# B&R Automation Studio project PrzewijarkaBRPraktyki (part 2)

#### RecipeMenage.st
```iecst
ACTION actRecipeManage:

		//Call TableConfiguration Variable
		RecipeControl.TableControl.Config;

		// create default recipes in case they don't exist yet on the target
		// recipes are created by using the the MpRecipeXml instance interface

		CASE RecipeCreateStep OF
			IDLE:

				IF MpRecepieXml_0.Active = TRUE AND MpRecipeUI_0.Active = TRUE THEN

				RecipeCreateStep 			:= CREATE_1;

				END_IF

			CREATE_1:	// create the first recipe with default values, file name and a known picture index (Bitmap Group in the HMI)
				MpRecepieXml_0.ErrorReset 			:= FALSE;

				gHMI.Recipe.CurrentRecipe.TensionLeft := 20;
				gHMI.Recipe.CurrentRecipe.TensionRight := 20;
				gHMI.Recipe.CurrentRecipe.Speed := 4;
				gHMI.Recipe.CurrentRecipe.Dencer1PID.P := 10;
				gHMI.Recipe.CurrentRecipe.Dencer1PID.I := 1;
				gHMI.Recipe.CurrentRecipe.Dencer2PID.P := 10;
				gHMI.Recipe.CurrentRecipe.Dencer2PID.I := 1;
				gHMI.Recipe.CurrentRecipe.RollLeft.MaxSize := 80;
				gHMI.Recipe.CurrentRecipe.RollLeft.MinSize := 30;
				gHMI.Recipe.CurrentRecipe.RollRight.MaxSize := 80;
				gHMI.Recipe.CurrentRecipe.RollRight.MinSize := 30;
				gHMI.Recipe.CurrentRecipe.DataRegistration := FALSE;

				MpRecepieXml_0.FileName 				:= ADR('mappRecipe1Test.xml');
				MpRecepieXml_0.Save					:= TRUE;
				RecipeCreateStep 					:= DONE_1;

			DONE_1:	// when CommandDone GoTo next step
				IF(MpRecepieXml_0.CommandDone) THEN
					RecipeCreateStep 			:= CREATE_2;
					MpRecepieXml_0.Save			:= FALSE;
				END_IF;

			CREATE_2:	// create the next recipe with default values, file name and a known picture index (Bitmap Group in the HMI)
				gHMI.Recipe.CurrentRecipe.TensionLeft := 40;
				gHMI.Recipe.CurrentRecipe.TensionRight := 40;
				gHMI.Recipe.CurrentRecipe.Speed := 8;
				gHMI.Recipe.CurrentRecipe.Dencer1PID.P := 10;
				gHMI.Recipe.CurrentRecipe.Dencer1PID.I := 1;
				gHMI.Recipe.CurrentRecipe.Dencer2PID.P := 10;
				gHMI.Recipe.CurrentRecipe.Dencer2PID.I := 1;
				gHMI.Recipe.CurrentRecipe.RollLeft.MaxSize := 80;
				gHMI.Recipe.CurrentRecipe.RollLeft.MinSize := 30;
				gHMI.Recipe.CurrentRecipe.RollRight.MaxSize := 80;
				gHMI.Recipe.CurrentRecipe.RollRight.MinSize := 30;
				gHMI.Recipe.CurrentRecipe.DataRegistration := FALSE;

				MpRecepieXml_0.FileName 			:= ADR('mappRecipe2Test.xml');
				MpRecepieXml_0.Save					:= TRUE;
				RecipeCreateStep 					:= DONE_2;

			DONE_2:	// when CommandDone GoTo next step
				IF (MpRecepieXml_0.CommandDone) THEN
					RecipeCreateStep 			:= CREATE_3;
					MpRecepieXml_0.Save			:= FALSE;
				END_IF;

			CREATE_3:	// create the next recipe with default values, file name and a known picture index (Bitmap Group in the HMI)

				gHMI.Recipe.CurrentRecipe.TensionLeft := 50;
				gHMI.Recipe.CurrentRecipe.TensionRight := 50;
				gHMI.Recipe.CurrentRecipe.Speed := 12;
				gHMI.Recipe.CurrentRecipe.Dencer1PID.P := 10;
				gHMI.Recipe.CurrentRecipe.Dencer1PID.I := 1;
				gHMI.Recipe.CurrentRecipe.Dencer2PID.P := 10;
				gHMI.Recipe.CurrentRecipe.Dencer2PID.I := 1;
				gHMI.Recipe.CurrentRecipe.RollLeft.MaxSize := 80;
				gHMI.Recipe.CurrentRecipe.RollLeft.MinSize := 30;
				gHMI.Recipe.CurrentRecipe.RollRight.MaxSize := 80;
				gHMI.Recipe.CurrentRecipe.RollRight.MinSize := 30;
				gHMI.Recipe.CurrentRecipe.DataRegistration := FALSE;

				MpRecepieXml_0.FileName 				:= ADR('mappRecipe3Test.xml');
				MpRecepieXml_0.Save					:= TRUE;
				RecipeCreateStep 					:= DONE_3;

			DONE_3:	// when CommandDone creating recipes is done
				IF(MpRecepieXml_0.CommandDone) THEN
					RecipeCreateStep 					:= CREATE_4;
					MpRecepieXml_0.Save					:= FALSE;
				END_IF;
			CREATE_4:	// create the next recipe with default values, file name and a known picture index (Bitmap Group in the HMI)

				gHMI.Recipe.CurrentRecipe.TensionLeft := 20;
				gHMI.Recipe.CurrentRecipe.TensionRight := 20;
				gHMI.Recipe.CurrentRecipe.Speed := 20;
				gHMI.Recipe.CurrentRecipe.Dencer1PID.P := 10;
				gHMI.Recipe.CurrentRecipe.Dencer1PID.I := 1;
				gHMI.Recipe.CurrentRecipe.Dencer2PID.P := 10;
				gHMI.Recipe.CurrentRecipe.Dencer2PID.I := 1;
				gHMI.Recipe.CurrentRecipe.RollLeft.MaxSize := 80;
				gHMI.Recipe.CurrentRecipe.RollLeft.MinSize := 30;
				gHMI.Recipe.CurrentRecipe.RollRight.MaxSize := 80;
				gHMI.Recipe.CurrentRecipe.RollRight.MinSize := 30;
				gHMI.Recipe.CurrentRecipe.DataRegistration := FALSE;

				MpRecepieXml_0.FileName 				:= ADR('mappRecipe4Test.xml');
				MpRecepieXml_0.Save					:= TRUE;
				RecipeCreateStep 					:= REFRESH;

			REFRESH:	// refresh the recipe list to make sure all the recipes are shown

				IF(MpRecepieXml_0.CommandDone) THEN
					RecipeCreateStep 					:= LOAD;
					MpRecepieXml_0	.Save					:= FALSE;
					UIConnect.Recipe.Refresh 	:= TRUE;
				END_IF;

			LOAD:	// load the first recipe to have a default recipe

				IF(UIConnect.Status = mpRECIPE_UI_STATUS_IDLE)THEN
					UIConnect.Recipe.Load 		:= TRUE;
					RecipeCreateStep 					:= DONE_4;
				END_IF

			DONE_4:	// if loading was successful the creation of the recipes is done

				IF(UIConnect.Status = mpRECIPE_UI_STATUS_IDLE)THEN
					RecipeCreateStep 			:= ALL_DONE;
					UIConnect.Recipe.Refresh 	:= FALSE;
					UIConnect.Recipe.Load 		:= FALSE;
				END_IF;

			ALL_DONE:

		END_CASE;

	//Edit Recipe
	IF RecipeControl.Edit.DialogOpen = TRUE THEN
		MaterialWidningEDITRecipe.TensionLeft := gHMI.Recipe.CurrentRecipe.TensionLeft;
		MaterialWidningEDITRecipe.TensionRight := gHMI.Recipe.CurrentRecipe.TensionRight;
		MaterialWidningEDITRecipe.Speed := gHMI.Recipe.CurrentRecipe.Speed;
		MaterialWidningEDITRecipe.Dencer1PID.P := gHMI.Recipe.CurrentRecipe.Dencer1PID.P;
		MaterialWidningEDITRecipe.Dencer1PID.I := gHMI.Recipe.CurrentRecipe.Dencer1PID.I;
		MaterialWidningEDITRecipe.Dencer2PID.P := gHMI.Recipe.CurrentRecipe.Dencer2PID.P;
		MaterialWidningEDITRecipe.Dencer2PID.I := gHMI.Recipe.CurrentRecipe.Dencer2PID.I;
		MaterialWidningEDITRecipe.RollLeft.MaxSize := gHMI.Recipe.CurrentRecipe.RollLeft.MaxSize;
		MaterialWidningEDITRecipe.RollLeft.MinSize := gHMI.Recipe.CurrentRecipe.RollLeft.MinSize;
		MaterialWidningEDITRecipe.RollRight.MaxSize := gHMI.Recipe.CurrentRecipe.RollRight.MaxSize;
		MaterialWidningEDITRecipe.RollRight.MinSize := gHMI.Recipe.CurrentRecipe.RollRight.MinSize;
		MaterialWidningEDITRecipe.DataRegistration := gHMI.Recipe.CurrentRecipe.DataRegistration;
		RecipeControl.Edit.DialogOpen							:= FALSE;
	END_IF

	IF RecipeControl.Edit.SaveRecipe = TRUE THEN
		gHMI.Recipe.CurrentRecipe.TensionLeft := MaterialWidningEDITRecipe.TensionLeft;
		gHMI.Recipe.CurrentRecipe.TensionRight := MaterialWidningEDITRecipe.TensionRight;
		gHMI.Recipe.CurrentRecipe.Speed := MaterialWidningEDITRecipe.Speed;
		gHMI.Recipe.CurrentRecipe.Dencer1PID.P := MaterialWidningEDITRecipe.Dencer1PID.P;
		gHMI.Recipe.CurrentRecipe.Dencer1PID.I := MaterialWidningEDITRecipe.Dencer1PID.I;
		gHMI.Recipe.CurrentRecipe.Dencer2PID.P := MaterialWidningEDITRecipe.Dencer2PID.P;
		gHMI.Recipe.CurrentRecipe.Dencer2PID.I := MaterialWidningEDITRecipe.Dencer2PID.I;
		gHMI.Recipe.CurrentRecipe.RollLeft.MaxSize := MaterialWidningEDITRecipe.RollLeft.MaxSize;
		gHMI.Recipe.CurrentRecipe.RollLeft.MinSize := MaterialWidningEDITRecipe.RollLeft.MinSize;
		gHMI.Recipe.CurrentRecipe.RollRight.MaxSize := MaterialWidningEDITRecipe.RollRight.MaxSize;
		gHMI.Recipe.CurrentRecipe.RollRight.MinSize := MaterialWidningEDITRecipe.RollRight.MinSize;
		gHMI.Recipe.CurrentRecipe.DataRegistration := MaterialWidningEDITRecipe.DataRegistration;
		UIConnect.New.FileName := MpRecepieXml_0.Info.LastLoadedRecipe;
		UIConnect.New.Create := TRUE;
		IF (UIConnect.Status = mpRECIPE_UI_STATUS_IDLE) THEN
			UIConnect.New.Create := FALSE;
			RecipeControl.Edit.SaveRecipe := FALSE;
		END_IF;

	END_IF

END_ACTION
```

### Program Logical/HMI/AuditPage (IEC)

#### Variables.var
```iecst
VAR
	MpAuditTrail_0 : MpAuditTrail;
	MpAuditTrailUI_0 : MpAuditTrailUI;
	AuditUIConnect : MpAuditTrailUIConnectType;
	Export : BOOL;
	Timer : TON;
END_VAR
```

#### Main.st
```iecst
PROGRAM _INIT
	MpAuditTrail_0.MpLink := ADR(gAuditTrail);
	MpAuditTrail_0.DeviceName := ADR('DATA');
	MpAuditTrail_0.Enable := TRUE;

	MpAuditTrailUI_0.MpLink := ADR(gAuditTrail);
	MpAuditTrailUI_0.UIConnect := ADR(AuditUIConnect);
	MpAuditTrailUI_0.Enable := TRUE;
END_PROGRAM

PROGRAM _CYCLIC
	IF Export THEN
		MpAuditTrail_0.Export := TRUE;
		IF (MpAuditTrail_0.Export) AND (MpAuditTrail_0.CommandDone) THEN
			MpAuditTrail_0.Export := FALSE;
			Export := FALSE;
		END_IF

		IF MpAuditTrail_0.ArchiveAvailable THEN
			MpAuditTrail_0.ExportArchive := TRUE;
		ELSE
			MpAuditTrail_0.ExportArchive := FALSE;
		END_IF
	ELSE
		MpAuditTrail_0.Export := FALSE;
	END_IF;

	Timer();
	MpAuditTrail_0();
	MpAuditTrailUI_0();

	IF MpAuditTrail_0.Error THEN
		MpAuditTrail_0.ErrorReset := TRUE;
	ELSE
		MpAuditTrail_0.ErrorReset := FALSE;
	END_IF;

	IF MpAuditTrailUI_0.Error THEN
		MpAuditTrailUI_0.ErrorReset := TRUE;
	ELSE
		MpAuditTrailUI_0.ErrorReset := FALSE;
	END_IF;
END_PROGRAM

PROGRAM _EXIT
	MpAuditTrail_0.Enable := FALSE;
	MpAuditTrailUI_0.Enable := FALSE;
END_PROGRAM
```

### Program Logical/HMI/AlarmPage (IEC)

#### Variables.var
```iecst
VAR
	MpAlarmXCore_0 : MpAlarmXCore;
	MpAlarmXHistory_0 : MpAlarmXHistory;
	Style : STRING[80];
END_VAR
```

#### Main.st
```iecst
PROGRAM _INIT
	(* MpLink przekazujemy przez referencję ADR *)
	MpAlarmXCore_0(MpLink := ADR(gAlarmXCore), Enable := TRUE);
	MpAlarmXHistory_0(MpLink := ADR(gAlarmXHistory), Enable := TRUE, DeviceName := ADR('DATA'));

END_PROGRAM

PROGRAM _CYCLIC
	//Power supply alarm
	IF gHMI.ModuleOK.PowerSupply = FALSE THEN
	  MpAlarmXSet(gAlarmXCore, 'ModuleOKErrorPS');
	END_IF;
	IF gHMI.ModuleOK.PowerSupply THEN
		MpAlarmXReset(gAlarmXCore, 'ModuleOKErrorPS');
	END_IF;

	//Analog input alarm
	IF gHMI.ModuleOK.AnalogInput = FALSE THEN
		MpAlarmXSet(gAlarmXCore, 'ModuleOKErrorAI');
	END_IF;
	IF gHMI.ModuleOK.AnalogInput THEN
		MpAlarmXReset(gAlarmXCore, 'ModuleOKErrorAI');
	END_IF;

	//System bus transmitter alarm
	IF gHMI.ModuleOK.SystemBusTransmitter = FALSE THEN
		MpAlarmXSet(gAlarmXCore, 'ModuleOKErrorBT');
	END_IF;
	IF gHMI.ModuleOK.SystemBusTransmitter THEN
		MpAlarmXReset(gAlarmXCore, 'ModuleOKErrorBT');
	END_IF;

	//Control keypad alarm
	IF gHMI.ModuleOK.ControlKeypad = FALSE THEN
		MpAlarmXSet(gAlarmXCore, 'ModuleOKError4XP');
	END_IF;
	IF gHMI.ModuleOK.ControlKeypad THEN
		MpAlarmXReset(gAlarmXCore, 'ModuleOKError4XP');
	END_IF;

	//Left winder alarm
	IF gTensionLogic.Status.LeftWinderDiameter < 30.0 THEN
		MpAlarmXSet(gAlarmXCore, 'LeftWinderDiameterLow');
	END_IF;
	IF gTensionLogic.Status.LeftWinderDiameter >= 30.0 THEN
		MpAlarmXReset(gAlarmXCore, 'LeftWinderDiameterLow');
	END_IF;

	//Right winder alarm
	IF gTensionLogic.Status.RightWinderDiameter < 30.0 THEN
		MpAlarmXSet(gAlarmXCore, 'RightWinderDiameterLow');
	END_IF;
	IF gTensionLogic.Status.RightWinderDiameter >= 30.0 THEN
		MpAlarmXReset(gAlarmXCore, 'RightWinderDiameterLow');
	END_IF;

	IF gHMI.Alarms.PendingAlarms THEN
		Style := 'orange';
	ELSE
		Style := 'default';
	END_IF;

	MpAlarmXCore_0();
	MpAlarmXHistory_0();

	gHMI.Alarms.PendingAlarms := UDINT_TO_BOOL(MpAlarmXCore_0.PendingAlarms);

	IF MpAlarmXCore_0.Error THEN
		MpAlarmXCore_0.ErrorReset := TRUE;
	ELSE
		MpAlarmXCore_0.ErrorReset := FALSE;
	END_IF;

	IF MpAlarmXHistory_0.Error THEN
		MpAlarmXHistory_0.ErrorReset := TRUE;
	ELSE
		MpAlarmXHistory_0.ErrorReset := FALSE;
	END_IF;
END_PROGRAM

PROGRAM _EXIT
	(* W sekcji exit trzeba wywołać/wyłaczyć blok funkcyjny (Enable := FALSE) *)
	MpAlarmXCore_0.Enable := FALSE;
	MpAlarmXHistory_0.Enable := FALSE;
END_PROGRAM
```

### Program Logical/HMI/ChartsDataPage (IEC)

#### Main.st - Init, cyclic, exit code
```iecst
PROGRAM _INIT
	MpDataRecorder_0.MpLink := ADR(gDataRecorder);
	MpDataRecorder_0.Enable := TRUE;
	MpDataRecorder_0.DeviceName := ADR('DATA');
	MpDataRecorder_0.RecordMode := mpDATA_RECORD_MODE_VALUE;
	MpDataRegPar_0.MpLink := ADR(gDataRecorder);
	MpDataRegPar_0.PVName := ADR('gHMI.Charts.Axis1');
	MpDataRegPar_0.Unit := ADR('m/min');
	MpDataRegPar_0.Description := ADR('Axis1 speed');

	MpDataRegPar_1.MpLink := ADR(gDataRecorder);
	MpDataRegPar_1.PVName := ADR('gHMI.Charts.Axis2');
	MpDataRegPar_1.Unit := ADR('m/min');
	MpDataRegPar_1.Description := ADR('Axis2 speed');

	MpDataRegPar_2.MpLink := ADR(gDataRecorder);
	MpDataRegPar_2.PVName := ADR('gHMI.Charts.Axis3');
	MpDataRegPar_2.Unit := ADR('m/min');
	MpDataRegPar_2.Description := ADR('Axis3 speed');

	MpDataRegPar_3.MpLink := ADR(gDataRecorder);
	MpDataRegPar_3.PVName := ADR('gHMI.Charts.Dancer1');
	MpDataRegPar_3.Unit := ADR('mm');
	MpDataRegPar_3.Description := ADR('Dancer 1 position');

	MpDataRegPar_4.MpLink := ADR(gDataRecorder);
	MpDataRegPar_4.PVName := ADR('gHMI.Charts.Dancer2');
	MpDataRegPar_4.Unit := ADR('mm');
	MpDataRegPar_4.Description := ADR('Dancer 2 position');

END_PROGRAM

PROGRAM _CYCLIC
	IF gHMI.Recipe.CurrentRecipe.DataRegistration THEN
		MpDataRecorder_0.Enable := TRUE;
		MpDataRecorder_0.Record := TRUE;
	ELSE
		MpDataRecorder_0.Enable := FALSE;
		MpDataRecorder_0.Record := FALSE;
	END_IF;

	IF gHMI.Charts.Record.Axis1 THEN
		MpDataRegPar_0.Enable := TRUE;
	ELSE
		MpDataRegPar_0.Enable := FALSE;
	END_IF;

	IF gHMI.Charts.Record.Axis2 THEN
		MpDataRegPar_1.Enable := TRUE;
	ELSE
		MpDataRegPar_1.Enable := FALSE;
	END_IF;

	IF gHMI.Charts.Record.Axis3 THEN
		MpDataRegPar_2.Enable := TRUE;
	ELSE
		MpDataRegPar_2.Enable := FALSE;
	END_IF;

	IF gHMI.Charts.Record.Dancer1 THEN
		MpDataRegPar_3.Enable := TRUE;
	ELSE
		MpDataRegPar_3.Enable := FALSE;
	END_IF;

	IF gHMI.Charts.Record.Dancer2 THEN
		MpDataRegPar_4.Enable := TRUE;
	ELSE
		MpDataRegPar_4.Enable := FALSE;
	END_IF;

	MpDataRecorder_0();
	MpDataRegPar_0();
	MpDataRegPar_1();
	MpDataRegPar_2();
	MpDataRegPar_3();
	MpDataRegPar_4();

	IF gHMI.Recipe.CurrentRecipe.DataRegistration THEN
		gHMI.Data.isSaving := 'TRUE';
	ELSE
		gHMI.Data.isSaving := 'FALSE';
	END_IF;

	IF MpDataRecorder_0.Error THEN
		MpDataRecorder_0.ErrorReset := TRUE;
	ELSE
		MpDataRecorder_0.ErrorReset := FALSE;
	END_IF;

	IF MpDataRegPar_0.Error THEN
		MpDataRegPar_0.ErrorReset := TRUE;
	ELSE
		MpDataRegPar_0.ErrorReset := FALSE;
	END_IF;

	IF MpDataRegPar_1.Error THEN
		MpDataRegPar_1.ErrorReset := TRUE;
	ELSE
		MpDataRegPar_1.ErrorReset := FALSE;
	END_IF;

	IF MpDataRegPar_2.Error THEN
		MpDataRegPar_2.ErrorReset := TRUE;
	ELSE
		MpDataRegPar_2.ErrorReset := FALSE;
	END_IF;

	IF MpDataRegPar_3.Error THEN
		MpDataRegPar_3.ErrorReset := TRUE;
	ELSE
		MpDataRegPar_3.ErrorReset := FALSE;
	END_IF;

	IF MpDataRegPar_4.Error THEN
		MpDataRegPar_4.ErrorReset := TRUE;
	ELSE
		MpDataRegPar_4.ErrorReset := FALSE;
	END_IF;
END_PROGRAM

PROGRAM _EXIT
	MpDataRecorder_0.Enable := FALSE;
	MpDataRegPar_0.Enable := FALSE;
	MpDataRegPar_1.Enable := FALSE;
	MpDataRegPar_2.Enable := FALSE;
	MpDataRegPar_3.Enable := FALSE;
	MpDataRegPar_4.Enable := FALSE;
END_PROGRAM
```

#### Types.typ - Local data types
```iecst
TYPE
	ChartsType : 	STRUCT
		Dancer1 : REAL;
		Dancer2 : REAL;
		Vtape : REAL;
		Axis1 : REAL;
		Axis2 : REAL;
		Axis3 : REAL;
	END_STRUCT;
END_TYPE
```

#### Variables.var - Local variables
```iecst
VAR
	MpDataRecorder_0 : MpDataRecorder;
	MpDataRegPar_0 : MpDataRegPar;
	MpDataRegPar_1 : MpDataRegPar;
	MpDataRegPar_2 : MpDataRegPar;
	MpDataRegPar_3 : MpDataRegPar;
	MpDataRegPar_4 : MpDataRegPar;
END_VAR
(*Data .csv display*)
VAR
	MpRecepieXml_Data : MpRecipeXml;
	MpRecipeUI_Data : MpRecipeUI;
	UIConnectData : MpRecipeUIConnectType;
END_VAR
```

#### actDisplayFiles.st
```iecst
ACTION actDisplayFiles:
	MpRecepieXml_Data.Enable := TRUE;
	MpRecepieXml_Data.MpLink := ADR(MpLinkRecipes);
	MpRecepieXml_Data.DeviceName := ADR('DATA');

	MpRecipeUI_Data.Enable := TRUE;
	MpRecipeUI_Data.MpLink := ADR(MpLinkRecipes);
	MpRecipeUI_Data.UIConnect := ADR(UIConnectData);

	UIConnectData.Recipe.Filter := '*.csv';

	MpRecepieXml_Data();
	MpRecipeUI_Data();

END_ACTION
```

### Program Logical/HMI/MainPage (IEC)

#### Main.st - Init, cyclic, exit code
```iecst
PROGRAM _INIT
	(* Insert code here *)

END_PROGRAM

PROGRAM _CYCLIC
	IF gTensionLogic.Status.EnableAxis1 = FALSE OR gTensionLogic.Status.EnableAxis2 = FALSE OR gTensionLogic.Status.EnableAxis3 = FALSE THEN
		aBORT := TRUE;
	END_IF;

	PhysicalBtn.Manual.ManProd := FALSE;
	gHMI.Recipe.EnableEditing := FALSE;

	IF Status.StateCurrent = 'Stopped'
	OR Status.StateCurrent = 'Aborted' THEN
		PhysicalBtn.Manual.ManProd := TRUE;
	END_IF;
	IF Status.StateCurrent = 'Idle'
	OR Status.StateCurrent = 'Stopped'
	OR Status.StateCurrent = 'Aborted' THEN
		gHMI.Recipe.EnableEditing := TRUE;
	END_IF;

	actBtnAssignment;
	actBasicColors;

	IF Status.ModeCurrent = 'Production' THEN
		actProdColors;
	END_IF;

	IF Status.ModeCurrent = 'Manual' THEN
		actManualMode;
	END_IF;

END_PROGRAM

PROGRAM _EXIT
	(* Insert code here *)

END_PROGRAM
```

#### Types.typ - Local data types
```iecst
TYPE
	ButtonStyles_type : 	STRUCT
		Start : STRING[80];
		Stop : STRING[80];
		Reset : STRING[80];
	END_STRUCT;
	ProductionBtn_type : 	STRUCT
		Start : Buttons_type;
		Stop : Buttons_type;
		Reset : Buttons_type;
	END_STRUCT;
	Buttons_type : 	STRUCT
		State : BOOL;
		ColorON : BOOL;
	END_STRUCT;
	PhysicalBtn_type : 	STRUCT
		Manual : ManualBtn_type;
		Production : ProductionBtn_type;
	END_STRUCT;
	ManualBtn_type : 	STRUCT
		Left : Buttons_type;
		Right : Buttons_type;
		ManProd : BOOL;
	END_STRUCT;
END_TYPE
```

#### Variables.var - Local variables
```iecst
VAR
	ButtonStyles : ButtonStyles_type;
	PhysicalBtn : PhysicalBtn_type;
	aBORT : BOOL;
END_VAR
```

#### actProdColors.st
```iecst
ACTION actProdColors:
	IF Status.StateCurrent = 'Idle' THEN
		ButtonStyles.Start := 'green';
		PhysicalBtn.Production.Start.ColorON := TRUE;
		ButtonStyles.Stop := 'red';
		PhysicalBtn.Production.Stop.ColorON := TRUE;
	END_IF;

	IF Status.StateCurrent = 'Starting'
		OR Status.StateCurrent = 'Execute'
		OR Status.StateCurrent = 'Completing'
		OR Status.StateCurrent = 'Complete'
		OR Status.StateCurrent = 'Resetting' THEN
		ButtonStyles.Stop := 'red';
		PhysicalBtn.Production.Stop.ColorON := TRUE;
	END_IF;

	IF Status.StateCurrent = 'Stopped'
		OR Status.StateCurrent = 'Complete'THEN
		ButtonStyles.Reset := 'blue';
		PhysicalBtn.Production.Reset.ColorON := TRUE;
	END_IF;
END_ACTION
```

#### actManualMode.st
```iecst
ACTION actManualMode:
	IF Status.StateCurrent = 'Stopped' THEN
		PhysicalBtn.Production.Reset.ColorON := TRUE;
		ButtonStyles.Reset := 'blue';
	END_IF;
	IF Status.StateCurrent = 'Idle' THEN
		PhysicalBtn.Production.Stop.ColorON := TRUE;
		ButtonStyles.Stop := 'red';
		actManualBtnAssignment;
	END_IF;
END_ACTION
```

#### actBasicColors.st
```iecst
ACTION actBasicColors:
	ButtonStyles.Start := 'default';
	ButtonStyles.Stop := 'default';
	ButtonStyles.Reset := 'default';
	PhysicalBtn.Production.Start.ColorON := FALSE;
	PhysicalBtn.Production.Stop.ColorON := FALSE;
	PhysicalBtn.Production.Reset.ColorON := FALSE;
END_ACTION
```

#### actBtnAssignment.st
```iecst
ACTION actBtnAssignment:
	gHMI.ControlBtn.Start := FALSE;
	gHMI.ControlBtn.Stop := FALSE;
	gHMI.ControlBtn.Reset := FALSE;
	IF PhysicalBtn.Production.Start.State = TRUE THEN
		gHMI.ControlBtn.Start := TRUE;
	END_IF;

	IF PhysicalBtn.Production.Stop.State = TRUE THEN
		gHMI.ControlBtn.Stop := TRUE;
	END_IF;

	IF PhysicalBtn.Production.Reset.State = TRUE THEN
		gHMI.ControlBtn.Reset := TRUE;
	END_IF;
END_ACTION
```

#### actManualBtnAssignment.st
```iecst
ACTION actManualBtnAssignment:
	IF PhysicalBtn.Manual.Left.State = TRUE OR gHMI.Manual.JogLeftRight.JogLeftTemp = TRUE THEN
		gHMI.Manual.JogLeftRight.JogLeft := TRUE;
		PhysicalBtn.Manual.Left.ColorON := TRUE;
	ELSE
		gHMI.Manual.JogLeftRight.JogLeft := FALSE;
		PhysicalBtn.Manual.Left.ColorON := FALSE;
	END_IF;
	IF PhysicalBtn.Manual.Right.State = TRUE OR gHMI.Manual.JogLeftRight.JogRightTemp = TRUE THEN
		gHMI.Manual.JogLeftRight.JogRight := TRUE;
		PhysicalBtn.Manual.Right.ColorON := TRUE;
	ELSE
		gHMI.Manual.JogLeftRight.JogRight := FALSE;
		PhysicalBtn.Manual.Right.ColorON := FALSE;
	END_IF;
END_ACTION
```

### Program Logical/HMI/DataPage

#### Variables.var
```iecst
VAR
	MpDataRecorder_0 : MpDataRecorder;
	StartRecording : BOOL;
	MpDataRegPar_0 : MpDataRegPar;
END_VAR
```

#### Main.st
```iecst
PROGRAM _INIT
	(* Insert code here *)
	MpDataRecorder_0.MpLink := ADR(gDataRecorder);
	MpDataRecorder_0.Enable := TRUE;
	MpDataRecorder_0.DeviceName := ADR('USER');
	MpDataRecorder_0.RecordMode := mpDATA_RECORD_MODE_TRIGGER;
	MpDataRecorder_0.Record := StartRecording;
	MpDataRecorder_0.Trigger := StartRecording;

	MpDataRegPar_0.MpLink := ADR(gDataRecorder);
	MpDataRegPar_0.Enable := TRUE;
	MpDataRegPar_0.PVName := ADR(StartRecording(*zmienna do monitorowania*));
END_PROGRAM

PROGRAM _CYCLIC
	(* Insert code here *)
	MpDataRecorder_0();
	MpDataRegPar_0();
END_PROGRAM

PROGRAM _EXIT
	(* Insert code here *)
	MpDataRecorder_0.Enable := FALSE;
	MpDataRegPar_0.Enable := FALSE;
END_PROGRAM
```

### actStopped.st
```iecst
ACTION actStopped:
	// wszystko wylaczamy
END_ACTION
```

### actAborting.st
```iecst
ACTION actAborting:

END_ACTION
```

### actAborted.st
```iecst
ACTION actAborted:

END_ACTION
```

### actClearing.st
```iecst
ACTION actClearing:
	// acknowlege all na liscie alarmow
END_ACTION
```

### actStopping.st
```iecst
ACTION actStopping:

END_ACTION
```

### actManIde.st - not listed in the package file held
```iecst
ACTION actManIdle:
	// odpalenie mozliwosci ruszania wszystkim
	// proponuje dwie opcje: 1 nawiajnie recznie ze sterowaniem trzema osiami
	// 						 2 ruszanie kazda z osi osobno
END_ACTION
```

### actManResetting.st - not listed in the package file held
```iecst
ACTION actManResetting:

END_ACTION
```

### actProductionIdle.st
```iecst
ACTION actProductionIdle:
	// czekanie na kolejny przycisk
END_ACTION
```

### actAutoExecute.st
```iecst
ACTION actExecute:

END_ACTION
```

### actAutoCompleting.st
```iecst
ACTION actAutoCompleting:

END_ACTION
```

### actAutoStarting.st
```iecst
ACTION actAutoStarting:

END_ACTION
```

### actAutoComplete.st
```iecst
ACTION actAutoComplete:

END_ACTION
```

### actAutoIdle.st
```iecst
ACTION actAutoIdle:

END_ACTION
```

### actAutoResetting.st
```iecst
ACTION actAutoResetting:

END_ACTION
```

### actCLEARING.st
```iecst
ACTION Action_9:

END_ACTION
```

Listed in the project but not available here: Logical/Global.typ, Logical/Global.var, Logical/PackMLCore/PackML/Types.typ, Logical/PackMLCore/PackML/Functions, Logical/Control/Tension/Dencers/DencersType.typ, Logical/Control/Axis/Axis1/Axis1/Axis1Type.typ, Logical/Control/Axis/Axis2/Axis2/Axis2.st, Logical/Control/Axis/Axis2/Axis2/Axis2Type.typ, Logical/Control/Axis/Axis3/Axis3/Axis3.st, Logical/Control/Axis/Axis3/Axis3/Axis3Type.typ, Logical/Control/SynMotion/SynMotion/SynMotionType.typ, Logical/Control/SynMotion/SynMotion/SynMotionVar.var, Logical/Main/ActionsPackML/Manual/actManIde.st, Logical/Main/ActionsPackML/Manual/actManResetting.st, Logical/Main/ActionsPackML/Production/actProductionExecute.st, Logical/Main/ActionsPackML/Production/actProductionCompleting.st, Logical/Main/ActionsPackML/Production/actProductionStarting.st, Logical/Main/ActionsPackML/Production/actProductionComplete.st, Logical/Main/ActionsPackML/Production/actProductionIdle.st, Logical/Main/ActionsPackML/Production/actProductionResetting.st, Logical/Documentation, Logical/Programs/gProgramsType.typ, Logical/Programs/gProgramsVar.var, Logical/Programs/ActionsPackML/Manual/actIdeMan.st, Logical/Programs/ActionsPackML/Manual/actResettingMan.st, Logical/Programs/Auto, Logical/Programs/Actions/actSTOPPED.st, Logical/Programs/Actions/actRESETTING.st, Logical/Programs/Actions/actIDLE.st, Logical/Programs/Actions/actSTARTING.st, Logical/Programs/Actions/actEXECUTE.st, Logical/Programs/Actions/actCOMPLETING.st, Logical/Programs/Actions/actCOMPLETE.st, Logical/Programs/Actions/actABORTING.st, Logical/Programs/Actions/actABORTED.st, Logical/Programs/Actions/actSTOPPING.st
